// TIA Portal V18 export
TYPE "SupplyFanChannel_v1"
// stored: IsFailsafeCompliant false
   STRUCT
      SAFSpeed1Ind : Array[0..2] of Bool;   // Off/On
      SAFSpeed2Ind : Array[0..2] of Bool;   // Off/On
      SAFIsBlockedByFrostProt : Array[0..2] of Bool;   // Off/On
   END_STRUCT;
END_TYPE
